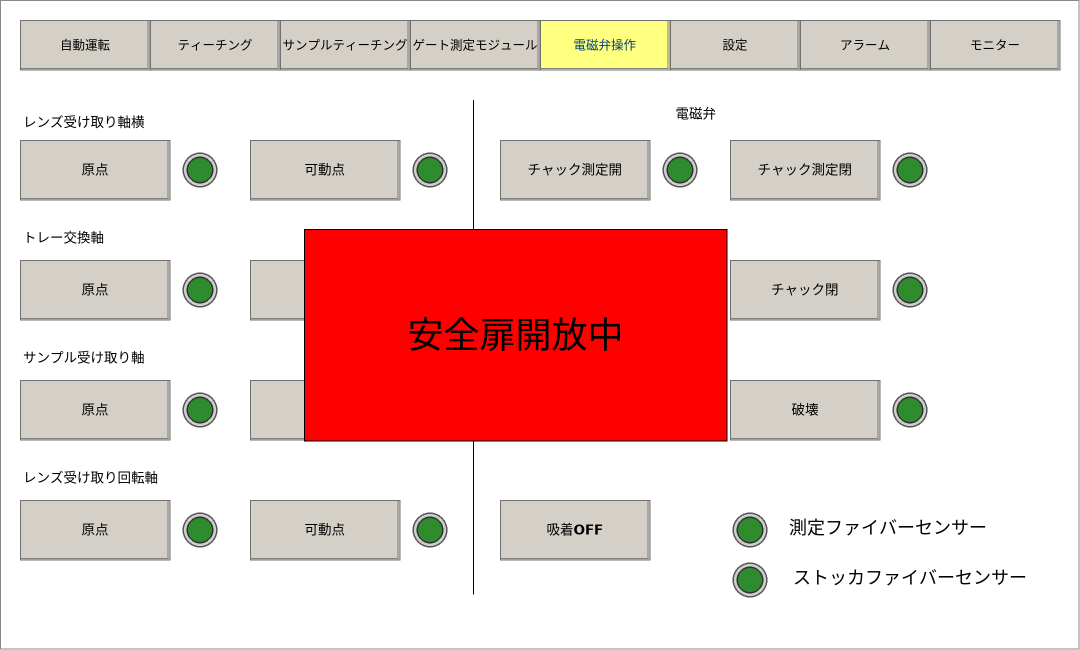
VISUALIZATION s_manual  // 1080x650
    Rectangle (0,0 1080x650)
    Button (20,140 150x60), "原点"
        tap gvl_visu.flg_btn_eleTransportNegative
    Button (20,260 150x60), "原点"
        tap gvl_visu.flg_btn_eleTrayChangeNegative
    Lamp1 (180,150 40x40), variable: gvl_elecylinder.ref_axis_transport.input.in_flg_sensA, style: Lamp-Lamp1-Green
    Lamp1 (180,270 40x40), variable: gvl_elecylinder.ref_axis_trayChange.input.in_flg_sensA, style: Lamp-Lamp1-Green
    Button (250,140 150x60), "可動点"
        tap gvl_visu.flg_btn_eleTransportPostive
    Button (250,260 150x60), "可動点"
        tap gvl_visu.flg_btn_eleTrayChangePositive
    Lamp1 (410,150 40x40), variable: gvl_elecylinder.ref_axis_transport.input.in_flg_sensB, style: Lamp-Lamp1-Green
    Lamp1 (410,270 40x40), variable: gvl_elecylinder.ref_axis_trayChange.input.in_flg_sensB, style: Lamp-Lamp1-Green
    Button (500,140 150x60), "チャック測定開"
        tap gvl_visu.flg_btn_svChuckOpen
    Button (500,260 150x60), "チャック開"
        tap gvl_visu.flg_btn_svPushOpen
    Button (730,260 150x60), "チャック閉"
        tap gvl_visu.flg_btn_svPushClose
    Lamp1 (890,150 40x40), tooltip "開", variable: gvl_solv.ref_chuck.in.in_flg_sensB, style: Lamp-Lamp1-Green
    Lamp1 (890,270 40x40), variable: gvl_solv.ref_push.in.in_flg_sensB, style: Lamp-Lamp1-Green
    Lamp1 (660,270 40x40), variable: gvl_solv.ref_push.in.in_flg_sensA, style: Lamp-Lamp1-Green
    Label (621,84 150x60), "電磁弁"
    Line (473,100) (473,594)
    Label (20,100 266x45), "レンズ受け取り軸横"
    Label (20,220 191x36), "トレー交換軸"
    Button (20,380 150x60), "原点"
        tap gvl_visu.flg_btn_eleSampleNegative
    Lamp1 (180,390 40x40), variable: gvl_elecylinder.ref_axis_sample.input.in_flg_sensA, style: Lamp-Lamp1-Green
    Button (250,380 150x60), "可動点"
        tap gvl_visu.flg_btn_eleSamplePositive
    Lamp1 (410,390 40x40), variable: gvl_elecylinder.ref_axis_sample.input.in_flg_sensB, style: Lamp-Lamp1-Green
    Label (20,340 262x36), "サンプル受け取り軸"
    Lamp1 (660,150 40x40), tooltip "開", variable: gvl_solv.ref_chuck.in.in_flg_sensA, style: Lamp-Lamp1-Green
    Label (20,460 262x36), "レンズ受け取り回転軸"
    Button (20,500 150x60), "原点"
        tap gvl_visu.flg_btn_eleRotaryNegative
    Lamp1 (180,510 40x40), variable: gvl_elecylinder.ref_axis_rotary.input.in_flg_sensA, style: Lamp-Lamp1-Green
    Button (250,500 150x60), "可動点"
        tap gvl_visu.flg_btn_eleRotaryPositive
    Lamp1 (410,510 40x40), variable: gvl_elecylinder.ref_axis_rotary.input.in_flg_sensB, style: Lamp-Lamp1-Green
    Button (730,140 150x60), "チャック測定閉"
        tap gvl_visu.flg_btn_svChuckClose
    Button (500,380 150x60), "吸着ON"
        tap gvl_visu.flg_btn_vacuumOn
    Button (730,380 150x60), "破壊"
        tap gvl_visu.flg_btn_breakOn
    Lamp1 (890,390 40x40), variable: gvl_solv.ref_ejector.input.in_flg_sensBrk, style: Lamp-Lamp1-Green
    Lamp1 (660,390 40x40), tooltip "開", variable: gvl_solv.ref_ejector.input.in_flg_sensVac, style: Lamp-Lamp1-Green
    Button (500,500 150x60), "吸着OFF"
        tap gvl_visu.flg_btn_vacuumOff
    Button (20,20 130x50), "自動運転"
        OnMouseClick: change screen: s_auto
    Button (150,20 130x50), "ティーチング"
        OnMouseClick: change screen: s_teaching1
    Button (670,20 130x50), "設定"
        OnMouseClick: change screen: s_setting
    Button (540,20 130x50), "電磁弁操作"
        OnMouseClick: change screen: s_manual
    Button (410,20 130x50), "ゲート測定モジュール"
        OnMouseClick: change screen: s_gm_teaching
    Button (800,20 130x50), "アラーム", colour toggle: gvl_io.flg_signalTowerRed
        OnMouseClick: change screen: s_alarm
    Button (280,20 130x50), "サンプルティーチング"
        OnMouseClick: change screen: s_alarm
    Rectangle (304,229 423x212), "安全扉開放中", text variable: gvl_io.flg_frontSaftyDoor or gvl_param.var_currentMode <> eP_programMode.auto, invisible if: gvl_io.flg_frontSaftyDoor or gvl_param.var_currentMode <> eP_programMode.auto
    Button (930,20 130x50), "モニター"
        OnMouseClick: change screen: s_monitor
    Lamp1 (730,510 40x40), variable: gvl_io.flg_gm_fiberSens, style: Lamp-Lamp1-Green
    Lamp1 (730,560 40x40), variable: gvl_io.flg_fiberSens, style: Lamp-Lamp1-Green
    Label (786,510 235x36), "測定ファイバーセンサー"
    Label (790,560 235x36), "ストッカファイバーセンサー"
END_VISUALIZATION

(* stored: Version 1.1.0.1, ProductVersion 3.1.4024.11
   Visu s_manual: Id {4f3dc8da-8db8-4e4e-9509-c35a358c6458} *)
